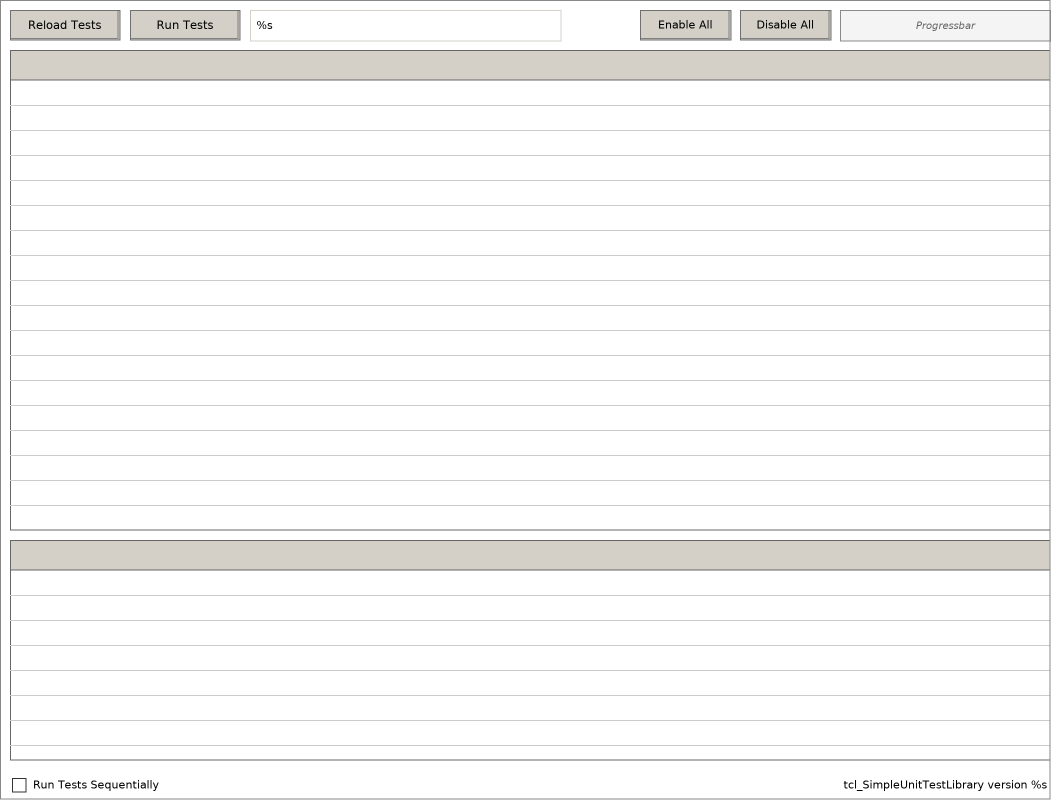
VISUALIZATION Visualization  // 1051x800
VAR_IN_OUT
    TestRunner : T_TestRunner;
    AssertionMessages : T_AssertionMessageList;
END_VAR
    Button (130,10 110x30), "Run Tests"
        OnMouseDown: execute { TestRunner.Reset := TRUE; }
        OnMouseUp: execute { TestRunner.Run := TRUE; }
    Textfield (250,10 311x31), "%s", text variable: TestRunner.ResultsSummary
    Progressbar (840,10 211x31), variable: TestRunner.TestsCompletedPercentage
    Rectangle (400,770 650x30), "tcl_SimpleUnitTestLibrary version %s", text variable: Global_Version.stLibVersion_tcl_SimpleUnitTestLibrary.sVersion
    Table (10,540 1040x220), data array: AssertionMessages.Messages
        p3854506369: AssertionMessages.Messages[INDEX]
        p1892666644: TestRunner.AssertionMessages._Count
        p2232123230: Assertion Messages
        p1128707560: AssertionMessages.Count - 1
    Checkbox (10,770 261x30), "Run Tests Sequentially", variable: TestRunner.RunTestsSequentially
    Table (10,50 1040x480), data array: TestRunner.Tests
        p3854506369: TestRunner.Tests[INDEX].ImageRef
        p1892666644: TestRunner.Tests[INDEX].SuiteName
        p338671338: TestRunner.Tests[INDEX].TestEnabled
        p2170511999: TestRunner.Tests[INDEX].TestHasFailed
        p3723444502: TestRunner.Tests[INDEX].TestHasFinished
        p1218418051: TestRunner.Tests[INDEX].TestName
        p746581629: TestRunner.Tests[INDEX].TestState
        p1757482276: Result
        p1128707560: TestRunner.TestCount - 1
        p1137915858: TestRunner.SelectedRow
        p1822360349: TestRunner.RowIsSelected
    Button (640,10 91x30), "Enable All"
        tap TestRunner.EnableAllTests
    Button (740,10 91x30), "Disable All"
        tap TestRunner.DisableAllTests
    Button (10,10 110x30), "Reload Tests"
        tap TestRunner.ReloadTests
END_VISUALIZATION

(* stored: Version 1.1.0.1, ProductVersion 3.1.4024.6
   Visu Visualization: Id {deef92dd-c8d0-4c0a-b471-21d2af44be99} *)
